(* CODESYS project 信号機_駅制御_北佐津.project

Project tree, tasks and I/O mapping:
  Device : CODESYS Control Win V3 x64, 3S - Smart Software Solutions GmbH, version 3.5.11.40
    application Application
      libraries: Standard, * (System); File Access, 3.5.7.0 (3S - Smart Software Solutions GmbH); Network, 3.5.7.0 (3S - Smart Software Solutions GmbH)
      task MainTask (cyclic, interval 4 ms, priority 0) calls EtherCAT_Master.EtherCAT_Task [EtherCAT_Master.EtherCAT_Task], StationControlMain
      function DecodeSwitchLeverOne [ST]
      program StationControlMain [ST]
      function block OnOffDelay [ST]
      function block TrainDetection [ST]
      SignalControl/
        function block FourStateSignal [ST]
        function block FourStateSignalDecoder [ST]
        function block ThreeStateSignal [ST]
        function block ThreeStateSignalDecoder [ST]
      declarations NVL_StationControl
      global variables NVL_StationStatus
      global variables ControlLever
      function block Decode_Levers [ST]
      function DecodeSignalLeverOne [ST]
      function block SwitchControl [ST]
      function block SignalControl [ST]
      function block Encode_Status [ST]
      function EncodeStatusOne [ST]
      function EncodeDetectionOne [ST]
    EtherCAT_Master : EtherCAT Master, 3S - Smart Software Solutions GmbH, version 3.5.11.40
        settings: NetworkName = 'イーサネット'; NetworkName = "イーサネット"; SrcAddress1 = 60449; SrcAddress2 = 3851182877
      NX_ECC202 : NX-ECC202 EtherCAT coupler V1.2, OMRON Corporation, order no. NX-ECC202, version Revision=16#00010002
          settings: ModularDevice = True; Number of Outputs = 0; Number of Infos about Outputs = 0; MDP_InputOffsets = [0,0,0,0,272]; MDP_OutputOffsets = [0,0,32,64,0]; StationAlias = 0; Sync.Length = 12; Sync.Length = 38; FMMU.Length = 12; FMMU.Length = 38; Number of RxPDOs of the Slave = 3; Number of TxPDOs of the Slave = 4; DC sync0 cycletime = 4000; DC sync1 cycletime = 4000; Number of SDO = 1; RxTxPdo.NumberofExcludes = 0; RxTxPdo.NumberofEntries = 1; RxTxPdo.Index = 16#1600; RxTxPdo.Fixed = True; RxTxPdo.Mandatory = True; RxTxPdo.Virtual = False; RxTxPdo.Sm = 2; RxTxPdo.Su = 0; RxTxPdo.Name = 'Output Data Set 1'; RxTxPdo.DependOnSlot = True; RxTxPdo.DependOnSlotGroup = False; RxTxPdo.OverwrittenByModule = True; Output Bit 32 bits.Index = 16#7003; Output Bit 32 bits.SubIndex = 1; Output Bit 32 bits.Size = 32; Output Bit 32 bits.Offset = 0; Output Bit 32 bits.DependOnSlot = True; Output Bit 32 bits.DependOnSlotGroup = True; RxTxPdo.NumberofExcludes = 0; RxTxPdo.NumberofEntries = 1; RxTxPdo.Index = 16#1604; RxTxPdo.Fixed = True; RxTxPdo.Mandatory = True; RxTxPdo.Virtual = False; RxTxPdo.Sm = 2;
            RxTxPdo.Su = 0; RxTxPdo.Name = 'Output Data Set 1'; RxTxPdo.DependOnSlot = True; RxTxPdo.DependOnSlotGroup = False; RxTxPdo.OverwrittenByModule = True; Output Bit 32 bits.Index = 16#7023; Output Bit 32 bits.SubIndex = 1; Output Bit 32 bits.Size = 32; Output Bit 32 bits.Offset = 0; Output Bit 32 bits.DependOnSlot = True; Output Bit 32 bits.DependOnSlotGroup = True; RxTxPdo.NumberofExcludes = 0; RxTxPdo.NumberofEntries = 1; RxTxPdo.Index = 16#1608; RxTxPdo.Fixed = True; RxTxPdo.Mandatory = True; RxTxPdo.Virtual = False; RxTxPdo.Sm = 2; RxTxPdo.Su = 0; RxTxPdo.Name = 'Output Data Set 1'; RxTxPdo.DependOnSlot = True; RxTxPdo.DependOnSlotGroup = False; RxTxPdo.OverwrittenByModule = True; Output Bit 32 bits.Index = 16#7043; Output Bit 32 bits.SubIndex = 1; Output Bit 32 bits.Size = 32; Output Bit 32 bits.Offset = 0; Output Bit 32 bits.DependOnSlot = True; Output Bit 32 bits.DependOnSlotGroup = True; RxTxPdo.NumberofExcludes = 0; RxTxPdo.NumberofEntries = 2; RxTxPdo.Index = 16#1BF8; RxTxPdo.Fixed = False; RxTxPdo.Mandatory = False; RxTxPdo.Virtual = False; RxTxPdo.Sm = 3; RxTxPdo.Su = 3; RxTxPdo.Name = '505th transmit PDO Mapping'; RxTxPdo.DependOnSlot = False; RxTxPdo.DependOnSlotGroup = False;
            RxTxPdo.OverwrittenByModule = False; NX Unit Registration Status 125.Index = 16#3003; NX Unit Registration Status 125.SubIndex = 4; NX Unit Registration Status 125.Size = 128; NX Unit Registration Status 125.Offset = 0; NX Unit Registration Status 125.DependOnSlot = False; NX Unit Registration Status 125.DependOnSlotGroup = False; NX Unit I/O Data Active Status 125.Index = 16#3006; NX Unit I/O Data Active Status 125.SubIndex = 4; NX Unit I/O Data Active Status 125.Size = 128; NX Unit I/O Data Active Status 125.Offset = 0; NX Unit I/O Data Active Status 125.DependOnSlot = False; NX Unit I/O Data Active Status 125.DependOnSlotGroup = False; RxTxPdo.NumberofExcludes = 0; RxTxPdo.NumberofEntries = 1; RxTxPdo.Index = 16#1BFF; RxTxPdo.Fixed = True; RxTxPdo.Mandatory = False; RxTxPdo.Virtual = False; RxTxPdo.Sm = 3; RxTxPdo.Su = 3; RxTxPdo.Name = '512th transmit PDO Mapping'; RxTxPdo.DependOnSlot = False; RxTxPdo.DependOnSlotGroup = False; RxTxPdo.OverwrittenByModule = False; Sysmac Error Status.Index = 16#2002; Sysmac Error Status.SubIndex = 1; Sysmac Error Status.Size = 8; Sysmac Error Status.Offset = 0; Sysmac Error Status.DependOnSlot = False; Sysmac Error Status.DependOnSlotGroup = False; RxTxPdo.NumberofExcludes = 0; RxTxPdo.NumberofEntries = 1; RxTxPdo.Index = 16#1BF4; RxTxPdo.Fixed = True; RxTxPdo.Mandatory = False; RxTxPdo.Virtual = False; RxTxPdo.Sm = 3; RxTxPdo.Su = 3; RxTxPdo.Name = '501st transmit PDO Mapping';
            RxTxPdo.DependOnSlot = False; RxTxPdo.DependOnSlotGroup = False; RxTxPdo.OverwrittenByModule = False; Entry.Offset = 0; Entry.DependOnSlot = False; Entry.DependOnSlotGroup = False; RxTxPdo.NumberofExcludes = 0; RxTxPdo.NumberofEntries = 1; RxTxPdo.Index = 16#1A0C; RxTxPdo.Fixed = True; RxTxPdo.Mandatory = True; RxTxPdo.Virtual = False; RxTxPdo.Sm = 3; RxTxPdo.Su = 0; RxTxPdo.Name = 'Input Data Set  1'; RxTxPdo.DependOnSlot = True; RxTxPdo.DependOnSlotGroup = False; RxTxPdo.OverwrittenByModule = True; Input Bit 32 bits.Index = 16#6063; Input Bit 32 bits.SubIndex = 1; Input Bit 32 bits.Size = 32; Input Bit 32 bits.Offset = 0; Input Bit 32 bits.DependOnSlot = True; Input Bit 32 bits.DependOnSlotGroup = True; Output Bit 32 bits.Name = 'Output Bit 32 bits'; Output Bit 32 bits.DataType = 'UDINT'; Output Bit 32 bits.Default = ''; Output Bit 32 bits.Comment = ''; Output Bit 32 bits.Name = 'Output Bit 32 bits'; Output Bit 32 bits.DataType = 'UDINT'; Output Bit 32 bits.Default = ''; Output Bit 32 bits.Comment = ''; Output Bit 32 bits.Name = 'Output Bit 32 bits'; Output Bit 32 bits.DataType = 'UDINT'; Output Bit 32 bits.Default = ''; Output Bit 32 bits.Comment = ''; NX Unit Registration Status 125.Name = 'NX Unit Registration Status 125'; NX Unit Registration Status 125.DataType = 'ARRAY [0..15] OF BYTE'; NX Unit Registration Status 125.Default = ''; NX Unit Registration Status 125.Comment = '';
            NX Unit I/O Data Active Status 125.Name = 'NX Unit I/O Data Active Status 125'; NX Unit I/O Data Active Status 125.DataType = 'ARRAY [0..15] OF BYTE'; NX Unit I/O Data Active Status 125.Default = ''; NX Unit I/O Data Active Status 125.Comment = ''; Sysmac Error Status.Name = 'Sysmac Error Status'; Sysmac Error Status.DataType = 'USINT'; Sysmac Error Status.Default = ''; Sysmac Error Status.Comment = ''; Entry.Default = ''; Input Bit 32 bits.Name = 'Input Bit 32 bits'; Input Bit 32 bits.DataType = 'UDINT'; Input Bit 32 bits.Default = ''; Input Bit 32 bits.Comment = ''
          unmapped channels: NX Unit Registration Status 125, NX Unit I/O Data Active Status 125, Sysmac Error Status, 
        NX_OD6121_5 : General output, OMRON Corporation, order no. NX-OD6121-5, version 0
            settings: Number of Outputs = 1; Number of Infos about Outputs = 1; Output Bit 32 bits.Offset = 0; Output Bit 32 bits.DependOnSlot = True; Output Bit 32 bits.DependOnSlotGroup = True; Output Bit 32 bits.Default = ''
            unmapped channels: Output Bit 32 bits
        NX_OD6121_5_1 : General output, OMRON Corporation, order no. NX-OD6121-5, version 0
            settings: Number of Outputs = 1; Number of Infos about Outputs = 1; Output Bit 32 bits.Index = 16#7023; Output Bit 32 bits.SubIndex = 1; Output Bit 32 bits.Size = 32; Output Bit 32 bits.Offset = 0; Output Bit 32 bits.DependOnSlot = True; Output Bit 32 bits.DependOnSlotGroup = True; Output Bit 32 bits.Name = 'Output Bit 32 bits'; Output Bit 32 bits.DataType = 'UDINT'; Output Bit 32 bits.Default = ''; Output Bit 32 bits.Comment = ''
            unmapped channels: Output Bit 32 bits
        NX_OD6121_5_2 : General output, OMRON Corporation, order no. NX-OD6121-5, version 0
            settings: Number of Outputs = 1; Number of Infos about Outputs = 1; Output Bit 32 bits.Index = 16#7043; Output Bit 32 bits.SubIndex = 1; Output Bit 32 bits.Size = 32; Output Bit 32 bits.Offset = 0; Output Bit 32 bits.DependOnSlot = True; Output Bit 32 bits.DependOnSlotGroup = True; Output Bit 32 bits.Name = 'Output Bit 32 bits'; Output Bit 32 bits.DataType = 'UDINT'; Output Bit 32 bits.Default = ''; Output Bit 32 bits.Comment = ''
            unmapped channels: Output Bit 32 bits
        NX_ID6142_5_1 : General input, OMRON Corporation, order no. NX-ID6142-5, version 0
            settings: Number of Inputs = 1; Number of Infos about Inputs = 1; Input Bit 32 bits.Index = 16#6063; Input Bit 32 bits.SubIndex = 1; Input Bit 32 bits.Size = 32; Input Bit 32 bits.Offset = 0; Input Bit 32 bits.DependOnSlot = True; Input Bit 32 bits.DependOnSlotGroup = True; Input Bit 32 bits.Name = 'Input Bit 32 bits'; Input Bit 32 bits.DataType = 'UDINT'; Input Bit 32 bits.Default = ''; Input Bit 32 bits.Comment = ''
            unmapped channels: Input Bit 32 bits
  data type E_SIGNAL_STATUS
*)

// E_SIGNAL_STATUS
TYPE E_SIGNAL_STATUS :
(
	R_Stop, YY_Warnig, Y_Caution, YG_Slowdown, G_Go
);
END_TYPE

// Device/Application/NVL_StationControl
//このグローバル変数リストはネットワーク経由受信です。
//送信者: ファイル 'C:\Users\Tomonobu\Documents\home\CodesysProject\StationControl.gvl' からインポートされました
//プロトコル: UDP

{attribute 'qualified_only'}
VAR_GLOBAL
	singal_lever_status: ARRAY[0..15] OF UINT;
	switch_lever_nml: ARRAY[0..15] OF UINT;
	switch_lever_rev: ARRAY[0..15] OF UINT;
END_VAR

// Device/Application/NVL_StationStatus
{attribute 'qualified_only'}
VAR_GLOBAL
	signal_display: ARRAY[0..15] OF E_SIGNAL_STATUS;
	signal_satus: ARRAY[0..15] OF UINT;
	signal_locked_nml: ARRAY[0..15] OF UINT;
	singal_locked_rev: ARRAY[0..15] OF UINT;
	switch_status: ARRAY[0..15] OF UINT;
	switch_locked_nml: ARRAY[0..15] OF UINT;
	switch_locked_rev: ARRAY[0..15] OF UINT;
	section_status: ARRAY[0..15] OF UINT;
END_VAR

// Device/Application/ControlLever
{attribute 'qualified_only'}
VAR_GLOBAL
	Switch_31Nml: BOOL;
	Switch_21Nml: BOOL;
	Switch_31Rev: BOOL;
	Switch_21Rev: BOOL;
	Signal_2R: BOOL;
	Signal_3R: BOOL;
	Signal_4R: BOOL;
	Signal_5R: BOOL;
	Signal_2L: BOOL;
	Signal_3L: BOOL;
	Signal_4L: BOOL;
	Signal_5L: BOOL;
END_VAR

// Device/Application/StationControlMain
PROGRAM StationControlMain
VAR
	Detect_Sensor : TrainDetection; 
	Input_Decode  : Decode_Levers;
	Output_Encode : Encode_Status;
	abDetectInfo_All : ARRAY[0..15] OF BOOL;

	Signal_2R: SignalControl;
	Signal_3R: SignalControl;
	Signal_4R: SignalControl;
	Signal_5R: SignalControl;

	Signal_2L: SignalControl;
	Signal_3L: SignalControl;
	Signal_4L: SignalControl;
	Signal_5L: SignalControl;

	Switch_31: SwitchControl;
	Switch_21: SwitchControl;
	
	// 在線検知
	bExist_31T: BOOL;
	bExist_21T: BOOL;
	bExist_2RT: BOOL;
	bExist_5RT: BOOL;
	
	QX4: INT;
	bSwitchRevReq: STRING(INT#4);
END_VAR

Input_Decode();
Output_Encode(sig_2R:=Signal_2R, sig_3R:=Signal_3R, sig_4R:=Signal_4R, sig_5R:=Signal_5R,
	          sig_2L:=Signal_2L, sig_3L:=Signal_3L, sig_4L:=Signal_4L, sig_5L:=Signal_5L,
			  swt_31:=Switch_31, swt_21:=Switch_21, abDetect:=abDetectInfo_All);
Detect_Sensor(abDetect => abDetectInfo_All);

// 在線検知信号
bExist_31T := abDetectInfo_All[0];
bExist_21T := abDetectInfo_All[1];
bExist_2RT := abDetectInfo_All[2];
bExist_5RT := abDetectInfo_All[3];

// 鎖錠信号
// 2L, 3L
IF Signal_2R.bLockActive OR
	Signal_4R.bLockActive OR
	Signal_5R.bLockActive OR
	NOT Switch_31.bStatusNormal OR
	NOT Switch_21.bStatusNormal THEN
	Signal_2L.bLockedNml := TRUE;
ELSE
	Signal_2L.bLockedNml := FALSE;
END_IF

//3L
IF Signal_3R.bLockActive OR
	Signal_4R.bLockActive OR
	Signal_5R.bLockActive OR
	Signal_5L.bLockActive OR
	Switch_31.bStatusNormal OR 
	Switch_21.bStatusNormal THEN
	Signal_3L.bLockedNml := TRUE;
ELSE
	Signal_3L.bLockedNml := FALSE;
END_IF

// 2R, 3R
IF Signal_2L.bLockActive OR
	Signal_3L.bLockActive THEN
	// 信号機で鎖錠
	Signal_2R.bLockedNml := TRUE;
	Signal_3R.bLockedNml := TRUE;
ELSE
	// 信号機の鎖錠解除(ポイントの鎖錠条件)
	IF Switch_21.bStatusNormal THEN
		Signal_2R.bLockedNml := FALSE;
	ELSE
		Signal_2R.bLockedNml := TRUE;
	END_IF
	IF NOT Switch_21.bStatusNormal THEN
		Signal_3R.bLockedNml := FALSE;
	ELSE
		Signal_3R.bLockedNml := TRUE;
	END_IF
END_IF

// 4R
IF Signal_4L.bLockActive OR
	Signal_2L.bLockActive OR
	Signal_3L.bLockActive OR
	NOT Switch_31.bStatusNormal OR
	NOT Switch_21.bStatusNormal THEN
	Signal_4R.bLockedNml := TRUE;
ELSE
	Signal_4R.bLockedNml := FALSE;
END_IF

// 5R
IF Signal_5L.bLockActive OR
	Signal_2L.bLockActive OR
	Signal_3L.bLockActive OR
	Signal_3R.bLockActive OR
	Switch_31.bStatusNormal OR
	Switch_21.bStatusNormal THEN
	Signal_5R.bLockedNml := TRUE;
ELSE
	Signal_5R.bLockedNml := FALSE;
END_IF

// 4L, 5L
IF Signal_4R.bLockActive OR
	Signal_5R.bLockActive THEN
	Signal_4L.bLockedNml := TRUE;
	Signal_5L.bLockedNml := TRUE;
ELSE
	// 信号機の鎖錠解除(ポイントの鎖錠条件)
	IF Switch_31.bStatusNormal THEN
		Signal_4L.bLockedNml := FALSE;
	ELSE
		Signal_4L.bLockedNml := TRUE;
	END_IF
	IF NOT Switch_31.bStatusNormal THEN
		Signal_5L.bLockedNml := FALSE;
	ELSE
		Signal_5L.bLockedNml := TRUE;
	END_IF
END_IF

// 31
IF Signal_2L.bLockActive OR
	Signal_4L.bLockActive OR
	Signal_4R.bLockActive THEN
	Switch_31.bLockedNml := TRUE;
ELSE
	Switch_31.bLockedNml := FALSE;
END_IF

IF Signal_3L.bLockActive OR
	Signal_5L.bLockActive OR
	Signal_5R.bLockActive THEN
	Switch_31.bLockedRev := TRUE;
ELSE
	Switch_31.bLockedRev := FALSE;
END_IF

// 21
IF Signal_4R.bLockActive OR
	Signal_2R.bLockActive OR
	Signal_2L.bLockActive THEN
	Switch_21.bLockedNml := TRUE;
ELSE
	Switch_21.bLockedNml := FALSE;
END_IF

IF Signal_5R.bLockActive OR
	Signal_3R.bLockActive OR
	Signal_5L.bLockActive THEN
	Switch_21.bLockedRev := TRUE;
ELSE
	Switch_21.bLockedRev := FALSE;
END_IF

// 信号制御
Signal_2R.bDisplayControl := bExist_21T;
Signal_3R.bDisplayControl := bExist_21T;
Signal_4R.bDisplayControl := bExist_31T OR bExist_5RT;
Signal_5R.bDisplayControl := bExist_31T OR bExist_2RT;
Signal_2L.bDisplayControl := bExist_21T OR bExist_5RT;
Signal_3L.bDisplayControl := bExist_21T OR bExist_2RT;
Signal_4L.bDisplayControl := bExist_31T;
Signal_5L.bDisplayControl := bExist_31T;

// 信号機間の連動
Signal_2R.eNextSignalStatus := E_SIGNAL_STATUS.G_Go;
Signal_3R.eNextSignalStatus := E_SIGNAL_STATUS.G_Go;
Signal_4R.eNextSignalStatus := Signal_2R.eSignalStatus;
Signal_5R.eNextSignalStatus := Signal_3R.eSignalStatus;

Signal_2L.eNextSignalStatus := Signal_4L.eSignalStatus;
Signal_3L.eNextSignalStatus := Signal_5L.eSignalStatus;
Signal_4L.eNextSignalStatus := E_SIGNAL_STATUS.G_Go;
Signal_5L.eNextSignalStatus := E_SIGNAL_STATUS.G_Go;

// 転換条件
Signal_2R(bLeverNormal := ControlLever.Signal_2R);
Signal_3R(bLeverNormal := ControlLever.Signal_3R);
Signal_4R(bLeverNormal := ControlLever.Signal_4R);
Signal_5R(bLeverNormal := ControlLever.Signal_5R);

Signal_2L(bLeverNormal := ControlLever.Signal_2L);
Signal_3L(bLeverNormal := ControlLever.Signal_3L);
Signal_4L(bLeverNormal := ControlLever.Signal_4L);
Signal_5L(bLeverNormal := ControlLever.Signal_5L);

Switch_31(bSwitchNmlReq := ControlLever.Switch_31Nml,
			bSwitchRevReq := ControlLever.Switch_31Rev);
Switch_21(bSwitchNmlReq := ControlLever.Switch_21Nml,
			bSwitchRevReq := ControlLever.Switch_21Rev);

// 信号機出力
%QX0.0 := Signal_2R.bLightGreen;
%QX0.1 := Signal_2R.bLightYellow;
%QX0.2 := Signal_2R.bLightRed;

%QX0.4 := Signal_3R.bLightGreen;
%QX0.5 := Signal_3R.bLightYellow;
%QX0.6 := Signal_3R.bLightRed;

%QX1.0 := Signal_4R.bLightGreen;
%QX1.1 := Signal_4R.bLightYellow;
%QX1.2 := Signal_4R.bLightRed;

%QX1.4 := Signal_5R.bLightGreen;
%QX1.5 := Signal_5R.bLightYellow;
%QX1.6 := Signal_5R.bLightRed;

%QX2.0 := Signal_2L.bLightGreen;
%QX2.1 := Signal_2L.bLightYellow;
%QX2.2 := Signal_2L.bLightRed;

%QX2.4 := Signal_3L.bLightGreen;
%QX2.5 := Signal_3L.bLightYellow;
%QX2.6 := Signal_3L.bLightRed;

%QX3.3 := Signal_4L.bLightGreen;
%QX3.2 := Signal_4L.bLightYellow;
%QX3.1 := Signal_4L.bLightRed;

%QX3.7 := Signal_5L.bLightGreen;
%QX3.6 := Signal_5L.bLightYellow;
%QX3.5 := Signal_5L.bLightRed;
	
// 転轍機出力
IF Switch_31.bStatusNormal THEN
	%QX4.0 := TRUE;
ELSE
	%QX4.0 := FALSE;
END_IF

IF Switch_21.bStatusNormal THEN
	%QX4.1 := TRUE;
ELSE
	%QX4.1 := FALSE;
END_IF

// 信号機出力

END_PROGRAM

// Device/Application/TrainDetection
FUNCTION_BLOCK TrainDetection
VAR_INPUT
END_VAR
VAR_OUTPUT
	abDetect: ARRAY[0..15] OF BOOL;
END_VAR
VAR
	DetectDelayExec: ARRAY[0..15] OF OnOffDelay;
	dwIdx: INT;
END_VAR

DetectDelayExec[0](bIN := %IX36.0);
DetectDelayExec[1](bIN := %IX36.1);
DetectDelayExec[2](bIN := %IX36.2);
DetectDelayExec[3](bIN := %IX36.3);
DetectDelayExec[4](bIN := %IX36.4);
FOR dwIdx:=0 TO 15 DO
	abDetect[dwIdx] := DetectDelayExec[dwIdx].bOUT;
END_FOR

END_FUNCTION_BLOCK

// Device/Application/OnOffDelay
FUNCTION_BLOCK OnOffDelay
VAR_INPUT
	bIN: BOOL;
END_VAR
VAR_OUTPUT
	bOUT: BOOL;
END_VAR
VAR
	OffDelayTimer: Standard.TOF;
	OnDelayTimer: Standard.TON;
	bPrevOutput: BOOL;
END_VAR

OffDelayTimer(IN:=bIN, PT:=T#0.5S);
OnDelayTimer(IN:=bIN, PT:=T#0.5S);
IF bPrevOutput THEN
	bOUT := OffDelayTimer.Q;
ELSE
	bOUT := OnDelayTimer.Q;	
END_IF
bPrevOutput := bOUT;

END_FUNCTION_BLOCK

// Device/Application/Decode_Levers
FUNCTION_BLOCK Decode_Levers
VAR_INPUT
END_VAR
VAR_OUTPUT
END_VAR
VAR
END_VAR

ControlLever.Signal_2R := DecodeSignalLeverOne(NVL_StationControl.singal_lever_status[0]);
ControlLever.Signal_3R := DecodeSignalLeverOne(NVL_StationControl.singal_lever_status[1]);
ControlLever.Signal_4R := DecodeSignalLeverOne(NVL_StationControl.singal_lever_status[2]);
ControlLever.Signal_5R := DecodeSignalLeverOne(NVL_StationControl.singal_lever_status[3]);
ControlLever.Signal_2L := DecodeSignalLeverOne(NVL_StationControl.singal_lever_status[4]);
ControlLever.Signal_3L := DecodeSignalLeverOne(NVL_StationControl.singal_lever_status[5]);
ControlLever.Signal_4L := DecodeSignalLeverOne(NVL_StationControl.singal_lever_status[6]);
ControlLever.Signal_5L := DecodeSignalLeverOne(NVL_StationControl.singal_lever_status[7]);

ControlLever.Switch_31Nml := DecodeSwitchLeverOne(NVL_StationControl.switch_lever_nml[0]);
ControlLever.Switch_21Nml := DecodeSwitchLeverOne(NVL_StationControl.switch_lever_nml[1]);

ControlLever.Switch_31Rev := DecodeSwitchLeverOne(NVL_StationControl.switch_lever_rev[0]);
ControlLever.Switch_21Rev := DecodeSwitchLeverOne(NVL_StationControl.switch_lever_rev[1]);

END_FUNCTION_BLOCK

// Device/Application/DecodeSignalLeverOne
FUNCTION DecodeSignalLeverOne : BOOL
VAR_INPUT
	Datalink_Val: UINT;
END_VAR
VAR
END_VAR

IF Datalink_Val = 1 THEN
	DecodeSignalLeverOne := FALSE;
ELSE
	DecodeSignalLeverOne := TRUE;	
END_IF

END_FUNCTION

// Device/Application/DecodeSwitchLeverOne
FUNCTION DecodeSwitchLeverOne : BOOL
VAR_INPUT
	Datalink_Val: UINT;
END_VAR
VAR
END_VAR

IF Datalink_Val = 1 THEN
	DecodeSwitchLeverOne := TRUE;
ELSE
	DecodeSwitchLeverOne := FALSE;	
END_IF

END_FUNCTION

// Device/Application/Encode_Status
FUNCTION_BLOCK Encode_Status
VAR_INPUT
	sig_2R: SignalControl;
	sig_3R: SignalControl;
	sig_4R: SignalControl;
	sig_5R: SignalControl;

	sig_2L: SignalControl;
	sig_3L: SignalControl;
	sig_4L: SignalControl;
	sig_5L: SignalControl;

	swt_31: SwitchControl;
	swt_21: SwitchControl;	
	
	abDetect: ARRAY[0..15] OF BOOL;
END_VAR
VAR_OUTPUT
END_VAR
VAR
END_VAR

NVL_StationStatus.signal_satus[0] := EncodeStatusOne(sig_2R.bStatusNormal);
NVL_StationStatus.signal_satus[1] := EncodeStatusOne(sig_3R.bStatusNormal);
NVL_StationStatus.signal_satus[2] := EncodeStatusOne(sig_4R.bStatusNormal);
NVL_StationStatus.signal_satus[3] := EncodeStatusOne(sig_5R.bStatusNormal);
NVL_StationStatus.signal_satus[4] := EncodeStatusOne(sig_2L.bStatusNormal);
NVL_StationStatus.signal_satus[5] := EncodeStatusOne(sig_3L.bStatusNormal);
NVL_StationStatus.signal_satus[6] := EncodeStatusOne(sig_4L.bStatusNormal);
NVL_StationStatus.signal_satus[7] := EncodeStatusOne(sig_5L.bStatusNormal);

NVL_StationStatus.switch_status[0] := EncodeStatusOne(swt_31.bStatusNormal);
NVL_StationStatus.switch_status[1] := EncodeStatusOne(swt_21.bStatusNormal);

NVL_StationStatus.section_status[0] := EncodeDetectionOne(abDetect[0]);
NVL_StationStatus.section_status[1] := EncodeDetectionOne(abDetect[1]);
NVL_StationStatus.section_status[2] := EncodeDetectionOne(abDetect[2]);
NVL_StationStatus.section_status[3] := EncodeDetectionOne(abDetect[3]);

END_FUNCTION_BLOCK

// Device/Application/EncodeStatusOne
FUNCTION EncodeStatusOne : UINT
VAR_INPUT
	bIsNormal: BOOL;
END_VAR
VAR
END_VAR

IF bIsNormal THEN
	EncodeStatusOne := 0;
ELSE
	EncodeStatusOne := 1;
END_IF

END_FUNCTION

// Device/Application/EncodeDetectionOne
FUNCTION EncodeDetectionOne : UINT
VAR_INPUT
	bIsDetect: BOOL;
END_VAR
VAR
END_VAR

IF bIsDetect THEN
	EncodeDetectionOne := 1;
ELSE
	EncodeDetectionOne := 0;
END_IF

END_FUNCTION

// Device/Application/SignalControl
FUNCTION_BLOCK SignalControl
VAR_INPUT
	bLeverNormal: BOOL;
	bLockedNml: BOOL;
	bLockedRev: BOOL;
	bDisplayControl: BOOL;
	bRouteLock: BOOL;
	eNextSignalStatus: E_SIGNAL_STATUS;
	Decoder: ThreeStateSignalDecoder;
END_VAR
VAR_OUTPUT
	bLockActive: BOOL;
	bStatusNormal: BOOL;
	eSignalStatus: E_SIGNAL_STATUS;
	bLightGreen: BOOL;
	bLightYellow: BOOL;
	bLightRed: BOOL;
END_VAR
VAR
	bLeverPrev: BOOL;
	bLeverNmlReq: BOOL;
	bLeverRevReq: BOOL;
END_VAR

// 微分検出
IF bLeverNormal AND NOT bLeverPrev THEN
	bLeverNmlReq := TRUE;
ELSE
	bLeverNmlReq := FALSE;
END_IF

IF NOT bLeverNormal AND bLeverPrev THEN
	bLeverRevReq := TRUE;
ELSE
	bLeverRevReq := FALSE;
END_IF
bLeverPrev := bLeverNormal;


// 状態制御
IF bStatusNormal THEN
	// 定位(微分検出)
	IF bLeverRevReq THEN
		IF (NOT bLockedNml) THEN
			// 鎖錠されていない
			bStatusNormal := FALSE;
			bLockActive := TRUE;
		END_IF
	END_IF
ELSE 
	// 反位(状態で判別)
	//		スイッチを定位に戻すか、内方に進入したら状態を定位に戻す。
	IF bLeverNormal OR bDisplayControl THEN
		IF (NOT bLockedRev) THEN
			// 鎖錠されていない
			bStatusNormal := TRUE;
			bLockActive := FALSE;
		END_IF
	END_IF
END_IF


// 現示制御
IF bStatusNormal THEN
	eSignalStatus := E_SIGNAL_STATUS.R_Stop;
ELSIF bDisplayControl THEN
	eSignalStatus := E_SIGNAL_STATUS.R_Stop;
ELSE
	IF eNextSignalStatus = E_SIGNAL_STATUS.R_Stop THEN
		eSignalStatus := E_SIGNAL_STATUS.Y_Caution;
	ELSE
		eSignalStatus := E_SIGNAL_STATUS.G_Go;
	END_IF
END_IF

// デコード
Decoder(sSignalStatus:=eSignalStatus,bRed=>bLightRed, bYellow=>bLightYellow, bGreen=>bLightGreen);

END_FUNCTION_BLOCK

// Device/Application/SignalControl/ThreeStateSignalDecoder
FUNCTION_BLOCK ThreeStateSignalDecoder
VAR_INPUT
	sSignalStatus: E_SIGNAL_STATUS;
END_VAR
VAR_OUTPUT
	bRed:     BOOL;
	bYellow : BOOL;
	bGreen:   BOOL;
END_VAR
VAR
END_VAR

bYellow  := FALSE;
bRed     := FALSE;
bGreen   := FALSE;


IF sSignalStatus = R_Stop THEN
	bRed    := TRUE;
ELSIF sSignalStatus = Y_Caution THEN
	bYellow := TRUE;
ELSIF sSignalStatus = G_Go THEN
	bGreen  := TRUE;
END_IF

END_FUNCTION_BLOCK

// Device/Application/SwitchControl
FUNCTION_BLOCK SwitchControl
VAR_INPUT
	bSwitchNmlReq: BOOL;
	bSwitchRevReq: BOOL;
	bLockedNml: BOOL;
	bLockedRev: BOOL;
END_VAR
VAR_OUTPUT
	bStatusNormal: BOOL;
	bLockActive: BOOL;
END_VAR
VAR
END_VAR

IF bSwitchNmlReq THEN
	// 定位
	IF (NOT bLockedRev) THEN
		bStatusNormal := TRUE;
		bLockActive := FALSE;
	ELSE
		bStatusNormal := FALSE;
		bLockActive := TRUE;
	END_IF
END_IF

IF bSwitchRevReq THEN
	// 反位
	IF (NOT bLockedNml) THEN
		bStatusNormal := FALSE;
		bLockActive := FALSE;
	ELSE
		bStatusNormal := TRUE;
		bLockActive := FALSE;
	END_IF
END_IF

END_FUNCTION_BLOCK

// Device/Application/SignalControl/FourStateSignal
FUNCTION_BLOCK FourStateSignal
VAR_INPUT
	bExist: BOOL;
	sNextSignalStatus: E_SIGNAL_STATUS;
END_VAR
VAR_OUTPUT
	sSignalStatus: E_SIGNAL_STATUS;
END_VAR
VAR
END_VAR

IF  bExist THEN
	sSignalStatus := R_Stop;
ELSE
	CASE sNextSignalStatus OF
	R_Stop : sSignalStatus := Y_Caution;
	YY_Warnig : sSignalStatus := Y_Caution;
	Y_Caution : sSignalStatus := YG_Slowdown;
	ELSE
		sSignalStatus := G_Go;
	END_CASE
END_IF

END_FUNCTION_BLOCK

// Device/Application/SignalControl/FourStateSignalDecoder
FUNCTION_BLOCK FourStateSignalDecoder
VAR_INPUT
	sSignalStatus: E_SIGNAL_STATUS;
END_VAR
VAR_OUTPUT
	bDummy:   BOOL;
	bYellow1: BOOL;
	bRed:     BOOL;
	bYellow2:  BOOL;
	bGreen:   BOOL;
END_VAR
VAR
END_VAR

bYellow1 := FALSE;
bRed     := FALSE;
bYellow2 := FALSE;
bGreen   := FALSE;


IF sSignalStatus = R_Stop THEN
	bRed := TRUE;
ELSIF sSignalStatus = Y_Caution THEN
	bYellow2 := TRUE;
ELSIF sSignalStatus = YG_Slowdown THEN
	bYellow1 := TRUE;
	bGreen := TRUE;
ELSIF sSignalStatus = G_Go THEN
	bGreen := TRUE;
END_IF

END_FUNCTION_BLOCK

// Device/Application/SignalControl/ThreeStateSignal
FUNCTION_BLOCK ThreeStateSignal
VAR_INPUT
	bExist: BOOL;
	sNextSignalStatus: E_SIGNAL_STATUS;
END_VAR
VAR_OUTPUT
	sSignalStatus: E_SIGNAL_STATUS;
END_VAR
VAR
END_VAR

IF  bExist THEN
	sSignalStatus := R_Stop;
ELSE
	CASE sNextSignalStatus OF
	R_Stop    : sSignalStatus := Y_Caution;
	YY_Warnig : sSignalStatus := Y_Caution;
	ELSE
		sSignalStatus := G_Go;
	END_CASE
END_IF

END_FUNCTION_BLOCK
